FUNCTION_BLOCK FB_LoadScan
VAR_INPUT
	bEnable			:BOOL;
	iConvStatus		:BYTE;
	bAutomat		:BOOL;
	
	bResetCTU		:BOOL;		
	bSetVal			:WORD;			
END_VAR
VAR_OUTPUT
	bEnableReadyID	:BOOL;
	bRequestID		:BOOL;
	bCountNoRead	:WORD;		//Кол-во несчитываний
	bOverflowID		:BOOL;		//Переполнение счетчика несчитываний ID
END_VAR
VAR
	fbPulsRequest	:R_TRIG;
	bStartRequest	:BOOL;
	fbDelayRead		:TON;
	WaitingID		:TON;
	bNoRead			:BOOL;		//Несчитывание
	bWriteIDgood	:BOOL;
	fbPulsNoread 	:R_TRIG;
	CTU 			:CTU;		//Счетчик
END_VAR
VAR_IN_OUT	
	stLoad			:ST_LoadData;
	bReadScan		:BOOL;
	sInID			:STRING;
END_VAR


bStartRequest:= bEnable AND bAutomat AND (iConvStatus=2 OR iConvStatus=3);

bEnableReadyID 	R= NOT bStartRequest;
bRequestID 	   	R= NOT bStartRequest  OR bReadScan;
bNoRead 		R= NOT bStartRequest;
bWriteIDgood    R= NOT bStartRequest;

fbPulsRequest(CLK:=bStartRequest);
IF fbPulsRequest.Q THEN
	bRequestID:=TRUE;
	bReadScan:=FALSE;
END_IF

fbDelayRead(IN:=bReadScan, PT:=T#0.3S);

WaitingID(IN:= bRequestID , PT:=T#3S);
bNoRead S= WaitingID.Q ;

fbPulsNoread(CLK:=bNoRead);

CTU(CU:=fbPulsNoread.Q, RESET:=bResetCTU, PV:=bSetVal);
bCountNoRead:=CTU.CV;

IF bReadScan AND NOT (bCountNoRead>=bSetVal) THEN
	stLoad.sID:= sInID;
	
	IF stLoad.sID<>'' OR fbDelayRead.Q THEN	
		bWriteIDgood:=TRUE;
		bReadScan:=FALSE;
	END_IF	
END_IF
bEnableReadyID S= bWriteIDgood OR bNoRead;

IF iConvStatus=0 THEN
	stLoad.sID:= '';
	stLoad.sWeight:= '';
	sInID:='';
END_IF

(*IF bCountNoRead>=bSetVal THEN bOverflowID:=TRUE;
	ELSE bOverflowID:=FALSE;
END_IF*)

END_FUNCTION_BLOCK

(* stored: Version 1.1.0.1, ProductVersion 3.1.4024.4
   POU FB_LoadScan: Id {e6dd006e-bee5-4a08-9e6c-de19f2059279}, SpecialFunc None *)
